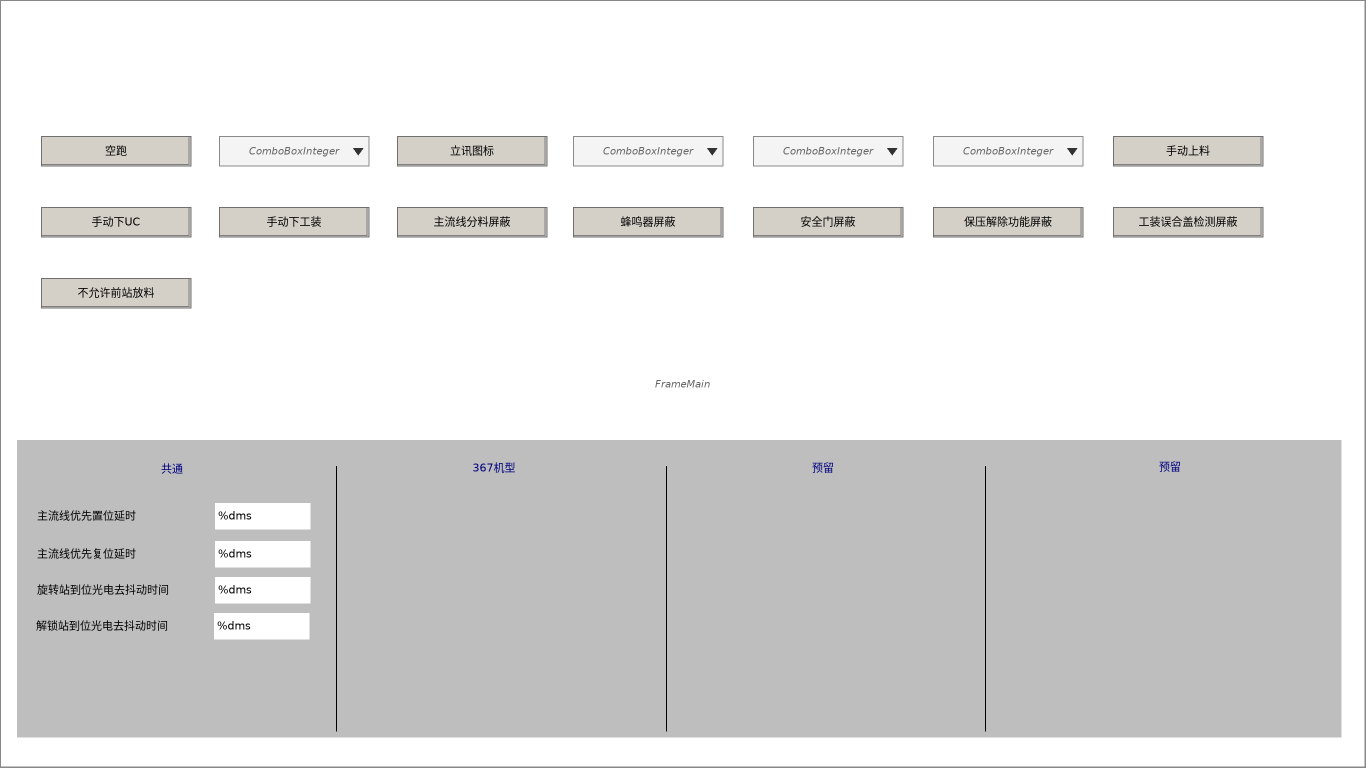
VISUALIZATION PageData  // 1366x768
    Frame (0,0 1366x768)
        shows FrameMain()
    Rectangle (16,439 1326x299)
    Button (41,136 150x30), "空跑"
        toggle GVL.stSetting.bDryRun
    ComboBoxInteger (219,136 150x30), variable: GVL_Data.stRecipe.eMachineType, text list: 'MachineType'
    Button (397,136 150x30), "立讯图标"
        toggle GVL_Data.stRecipe.bLuxshardict
    ComboBoxInteger (573,136 150x30), variable: GVL_Data.stRecipe.eLoadClose, text list: 'LineLoadClose'
    ComboBoxInteger (753,136 150x30), variable: GVL_Data.stRecipe.eProductType, text list: 'ProductType'
    Button (41,207 150x30), "手动下UC"
        toggle GVL.stSetting.bManualUnloadUc
    Button (219,207 150x30), "手动下工装"
        toggle GVL.stSetting.bManualUnloadFrock
    Button (1113,136 150x30), "手动上料"
        toggle GVL.stSetting.bManualLoad
    Button (397,207 150x30), "主流线分料屏蔽"
        toggle GVL.stSetting.bLine0BufferShield
    Button (573,207 150x30), "蜂鸣器屏蔽"
        toggle G_stSystem.stInput.bQuiet
    Button (753,207 150x30), "安全门屏蔽"
        toggle GVL.stSetting.bSafeDoorShield
    Button (933,207 150x30), "保压解除功能屏蔽"
        toggle GVL.stSetting.bOpenLockPressShield
    ComboBoxInteger (933,136 150x30), variable: GVL_Data.stRecipe.eLoadClass, text list: 'LineLoadClase'
    Button (41,278 150x30), "不允许前站放料"
        toggle GVL.stSetting.bStopFrontStation
    Button (1113,207 150x30), "工装误合盖检测屏蔽"
        toggle GVL.stSetting.bFrockCloseCheckShield
    RoundedRectangle (215,503 95x26), "%dms", text variable: GVL_Data.stRecipe.arrAutoTon[E_Timer.Line0PriorityOnDelay]
        OnMouseClick: write the text variable via Default
    Label (34,501 173x30), "主流线优先置位延时"
    RoundedRectangle (215,541 95x26), "%dms", text variable: GVL_Data.stRecipe.arrAutoTon[E_Timer.Line0PriorityOffDelay]
        OnMouseClick: write the text variable via Default
    Label (34,539 173x30), "主流线优先复位延时"
    Label (136,454 72x30), "共通"
    Label (458,453 72x30), "367机型"
    Line (336,466) (336,731)
    Line (666,466) (666,731)
    Label (787,453 72x30), "预留"
    Line (985,466) (985,731)
    Label (1134,452 72x30), "预留"
    RoundedRectangle (215,577 95x26), "%dms", text variable: GVL_Data.stRecipe.arrAutoTon[E_Timer.SteeringCheck1F]
        OnMouseClick: write the text variable via Default
    Label (34,575 173x30), "旋转站到位光电去抖动时间"
    RoundedRectangle (214,613 95x26), "%dms", text variable: GVL_Data.stRecipe.arrAutoTon[E_Timer.OpenLockCheckF]
        OnMouseClick: write the text variable via Default
    Label (33,611 173x30), "解锁站到位光电去抖动时间"
END_VISUALIZATION

(* stored: Version 1.1.0.1, ProductVersion 3.1.4024.3
   Visu PageData: Id {0b2b5a27-2634-4cb9-8f58-77bd32f946b4} *)
